FUNCTION "_sexagesimalToRadians" : Real
TITLE = {"version":"v1.0","author":"cyanezf","family":"core/converter","status":"current","deprecatedBy": null,"dependencies" : []}
{ S7_Optimized_Access := 'TRUE' }
AUTHOR : cyanezf
FAMILY : 'core/converter'
NAME : _sexagesimalToRadians
VERSION : 1.0

   VAR_INPUT
      angle : Real;   // Sexagesimal angle
   END_VAR

   VAR CONSTANT
      PI : Real := 3.141593;   // PI aproximation: 3.141 592 653 589 793 238
   END_VAR

BEGIN
(*--
# Documentation

## Log

| version | date | author | description |
|:-------:|:----:|:------:|:------------|
| v1.0 | 2023-06-06 | cyanezf | First version |

## Description

This funtions converts an sexagesimal angle to radian.

--*)

  // Return
	#_sexagesimalToRadians := #angle * #PI / 180.0;

  // Save RLO
	ENO := TRUE;

END_FUNCTION

